// TIA Portal V16 export
// export: Created 2025-05-30T16:36:22.9924756Z, ExportSetting WithDefaults, DisplayName Totally Integrated Automation Portal, DisplayVersion V16, DisplayName TIA Portal Version Control Interface, DisplayVersion V16, DisplayName TIA Portal Openness, DisplayVersion V16, DisplayName STEP 7 Professional, DisplayVersion V16, DisplayName STEP 7 Safety, DisplayVersion V16, DisplayName WinCC Advanced, DisplayVersion V16
DATA_BLOCK "2in-1out_Block_LED-Estop"   // DB1
VERSION : 0.1
// stored: AutoNumber true, InstanceOfName 2in-1out_Block, InstanceOfType FB
"2in-1out_Block"
   // VAR_INPUT
   //    "Input Contact 1" : Bool;
   //    "Input Contact 2" : Bool;
   // END_VAR
   // VAR_OUTPUT
   //    "Output Contact 1" : Bool;
   // END_VAR
BEGIN
END_DATA_BLOCK
